PROGRAM INTERNAL PRG_TEST_GLOBAL // A place to call global function blocks (singletons) that can be used by all tests

Sys_Variables.fbSystemVariables();
GVL_Utilities.fbFaultHandler();

END_PROGRAM

(* stored: Version 1.1.0.1, ProductVersion 3.1.4024.11
   POU PRG_TEST_GLOBAL: Id {df90b9c7-1da5-0652-2def-5bbda35b922b}, SpecialFunc None *)
